// Writes an sfixed64 value, without a tag, to the stream.
FUNCTION F_WriteSFixed64 : HRESULT
VAR_INPUT
    stBuffer    : ST_Span;
END_VAR
VAR_IN_OUT
    stState     : ST_WriterInternalState;
END_VAR
VAR_INPUT
    nValue : LINT;
END_VAR
VAR
END_VAR

F_WriteSFixed64 := F_WriteRawLittleEndian64(stBuffer, stState, TO_ULINT(nValue));

END_FUNCTION

(* stored: Version 1.1.0.1
   POU F_WriteSFixed64: Id {7b2a4de3-db7e-43cb-9133-2e939ff4fe38}, SpecialFunc None *)
